{attribute 'qualified_only'}
{attribute 'strict'}
TYPE state_enum :
(
	startup_mode,
	jog_joint_mode,
	jog_cartesian_mode,
	auto_mode,
	emg_stop_mode,
	comm_fault_mode,
	manual_mode
);
END_TYPE

(* stored: Version 1.1.0.1, ProductVersion 3.1.4024.13
   DUT state_enum: Id {ca274e56-8cfc-4bff-bb62-2057a3e7a0f5} *)
